{attribute 'linkalways'} 
{attribute 'no_explicit_call' := 'This FB is a CLASS and must be accessed using methods or properties'}
{attribute 'enable_dynamic_creation'}
FUNCTION_BLOCK Node_F_VN_UprightInnerRectangle EXTENDS VisionNode
VAR
    ipSrcImage : _ITcVnImage;
    stRectangle : _TcVnRectangle_DINT;
    hrPrev : _HRESULT(S_OK);
	hresult : _HRESULT(S_OK);
END_VAR

METHOD PUBLIC  Clone : I_Node
VAR
	pNode : POINTER TO Node_F_VN_UprightInnerRectangle;
END_VAR
pNode := __NEW(Node_F_VN_UprightInnerRectangle);
Clone := pNode^;
END_METHOD

METHOD FB_init : BOOL
VAR_INPUT
	bInitRetains : BOOL; // if TRUE, the retain variables are initialized (warm start / cold start)
	bInCopyCode : BOOL;  // if TRUE, the instance afterwards gets moved into the copy code (online change)
END_VAR
AddInput('ipSrcImage', ipSrcImage);
AddInput('hrPrev', hrPrev);
AddOutput('stRectangle', stRectangle);
AddOutput('hresult', hresult);
END_METHOD

METHOD PROTECTED OnExecute
hresult.Value := F_VN_UprightInnerRectangle(
	ipSrcImage := ipSrcImage.Value,
    stRectangle := stRectangle.Value,
	hrPrev:= hrPrev.Value);
END_METHOD

METHOD PUBLIC PreExecutionCheck
VAR_INPUT
	Check : I_PreExecutionChecks;
END_VAR
Check.IsTrue(ipSrcImage.IsValid, 'ipSrcImage must contain an image');
Check.IsTrue(ipSrcImage.IsPixelDepth(8), 'ipSrcImage must be 8 bit pixel depth');
Check.IsTrue(ipSrcImage.HasChannelCount(1), 'ipSrcImage must contain 1 channel');
END_METHOD

END_FUNCTION_BLOCK

(* stored: Version 1.1.0.1, ProductVersion 3.1.4024.15
   POU Node_F_VN_UprightInnerRectangle: Id {fb9b9e03-22c2-4fd0-a6a9-19607c58231f}, SpecialFunc None
   Folder Constructor: Id {87065cc1-a199-4df7-88f7-d014fd39b552}
   Method Clone: Id {ae2f98c1-ad0e-4215-a992-5c55987ac4ca}
   Method FB_init: Id {a5de9d6b-c0fc-4bb4-a67c-c3c6675333db}
   Method OnExecute: Id {d091774c-83d5-4e4a-a888-0079902430f0}
   Method PreExecutionCheck: Id {e99157c5-2094-4132-9a68-ee248cbb6327} *)
